PROGRAM MAIN
VAR
	fbAmpel : FB_Ampel;
	fbEZylinder1 : FB_EZylinder;
	fbEZylinder2 : FB_EZylinder;
	MCPowerBand : MC_Power;
	MCPowerDispenser1 	: MC_Power;
	MCPowerDispenser2 	: MC_Power;
	MCPowerDispenser3 	: MC_Power;
	MCPowerAchseX	 	: MC_Power;
	MCPowerAchseY 	: MC_Power;
	MCPowerAchseZ 	: MC_Power;
	MCPowerAchseG 	: MC_Power;
	fbAbfullModul : FB_Abfullmodul;
	fbRoboter : FB_Robotersteuerung;
	fbIotMqttCommunication : FB_IotMqttCommunication;
	
	nRoboterLagerIndex : INT;
	

	ix : REAL;
	ry : UINT;
	
	
  	

END_VAR

ry := TO_UINT(FUN_Scale(ix,4096, 0, 350, 0));

IFC_HW.ax_BandMotor.ReadStatus();
IFC_HW.ax_Extruder1.ReadStatus();
IFC_HW.ax_Extruder2.ReadStatus();
IFC_HW.ax_Extruder3.ReadStatus();



MCPowerBand(
	Axis:= IFC_HW.ax_BandMotor , 
	Enable:= TRUE , 
	Enable_Positive:= TRUE, 
	Enable_Negative:= TRUE, 
	Override:= , 
	BufferMode:= , 
	Options:= , 
	Status=> , 
	Busy=> , 
	Error=> , 
	ErrorID=> );
	
MCPowerDispenser1(
	Axis:= IFC_HW.ax_Extruder1, 
	Enable:= TRUE, 
	Enable_Positive:= TRUE, 
	Enable_Negative:= TRUE, 
	Override:= , 
	BufferMode:= , 
	Options:= , 
	Status=> , 
	Busy=> , 
	Error=> , 
	ErrorID=> );
	
MCPowerDispenser2(
	Axis:= IFC_HW.ax_Extruder2, 
	Enable:= TRUE, 
	Enable_Positive:= TRUE, 
	Enable_Negative:= TRUE, 
	Override:= , 
	BufferMode:= , 
	Options:= , 
	Status=> , 
	Busy=> , 
	Error=> , 
	ErrorID=> );
	
MCPowerDispenser3(
	Axis:= IFC_HW.ax_Extruder3, 
	Enable:= TRUE, 
	Enable_Positive:= TRUE, 
	Enable_Negative:= TRUE, 
	Override:= , 
	BufferMode:= , 
	Options:= , 
	Status=> , 
	Busy=> , 
	Error=> , 
	ErrorID=> );
	
MCPowerAchseX(
	Axis:= IFC_HW.ax_ManX, 
	Enable:= TRUE, 
	Enable_Positive:= TRUE, 
	Enable_Negative:= TRUE, 
	Override:= , 
	BufferMode:= , 
	Options:= , 
	Status=> , 
	Busy=> , 
	Error=> , 
	ErrorID=> );
	
MCPowerAchseY(
	Axis:= IFC_HW.ax_ManY, 
	Enable:= TRUE, 
	Enable_Positive:= TRUE, 
	Enable_Negative:= TRUE, 
	Override:= , 
	BufferMode:= , 
	Options:= , 
	Status=> , 
	Busy=> , 
	Error=> , 
	ErrorID=> );

MCPowerAchseZ(
	Axis:= IFC_HW.ax_ManZ, 
	Enable:= TRUE, 
	Enable_Positive:= TRUE, 
	Enable_Negative:= TRUE, 
	Override:= , 
	BufferMode:= , 
	Options:= , 
	Status=> , 
	Busy=> , 
	Error=> , 
	ErrorID=> );
	
MCPowerAchseG(
	Axis:= IFC_HW.ax_ManG, 
	Enable:= TRUE, 
	Enable_Positive:= TRUE, 
	Enable_Negative:= TRUE, 
	Override:= , 
	BufferMode:= , 
	Options:= , 
	Status=> , 
	Busy=> , 
	Error=> , 
	ErrorID=> );


fbAbfullModul(
	bEnable:= IFC_HW.bEnable, 
	bExecute:= IFC_HW.bExecute, 
	bBandSens1:= IFC_HW.bBandSens1, 
	bBandSens2:= IFC_HW.bBandSens2, 
	bBandSens3:= IFC_HW.bBandSens3, 
	bBandSens4:= IFC_HW.bBandSens4, 
	bEinzelSens1:= IFC_HW.bEinzelSens1 , 
	bEinzelSens2:= IFC_HW.bEinzelSens2, 
	bEinzelSens3:= IFC_HW.bEinzelSens3, 
	nLagerIndex:= , 
	bGate1=> fbEZylinder1.bGate, 
	bGate2=> fbEZylinder2.bGate, 
	bStopper1=> IFC_HW.bBandHub1 , 
	bStopper2=> IFC_HW.bBandHub2, 
	bStopper3=> IFC_HW.bBandHub3, 
	eState=> , 
	axFoerderband:= IFC_HW.ax_BandMotor, 
	axDispenser1:= IFC_HW.ax_Extruder1, 
	axDispenser2:= IFC_HW.ax_Extruder2, 
	axDispenser3:= IFC_HW.ax_Extruder3
 );
 
 fbRoboter(
    bEnable := IFC_HW.bEnable,
    bExecute := IFC_HW.bExecute,

    bSensBand4 := IFC_HW.bBandSens4,
    bSensEndX := IFC_HW.bManEndXmin,
    bSensEndY := IFC_HW.bManEndYmin,
    bSensEndZ := IFC_HW.bManEndZmin,
    bSensEndG := IFC_HW.bManEndGmin,

    eState => ,

    bBrakeZ => IFC_HW.bManBrakeZ,
    bGripperClosed => IFC_HW.bGripperClosed,

    axX := IFC_HW.ax_ManX,
    axY := IFC_HW.ax_ManY,
    axZ := IFC_HW.ax_ManZ,
    axG := IFC_HW.ax_ManG,

    nLagerIndex := nRoboterLagerIndex
);
 
 fbIotMqttCommunication(
	sTopicToPublish:= 'bEnable',
	sMessageToPublish:= BOOL_TO_STRING(IFC_HW.bEnable),
);
	
fbEZylinder1(bGate:= , bError:= ,
			 bR1=> IFC_HW.bR1AKT1, bR2=> IFC_HW.bR2AKT1);
fbEZylinder2(bGate:= , bError:= , 
			bR1=> IFC_HW.bR1AKT2, bR2=> IFC_HW.bR2AKT2 );
			
fbAmpel(eState:= fbAbfullmodul.eState, bAmpelGrun=> IFC_HW.bAmpelGrun, bAmpelRot=> IFC_HW.bAmpelRot , bAmpelGelb=> IFC_HW.bAmpelGelb);

END_PROGRAM

(* stored: Version 1.1.0.1, ProductVersion 3.1.4024.15
   POU MAIN: Id {e19b8e30-f99f-45cf-bb86-ad2b8de51b93}, SpecialFunc None *)
